{attribute addProperty BoxType "EP9128-0021-0018"}
{attribute addProperty Id "A_0013_EP9128_0021_0019A_0013_EP9128_0021_0019_07EDD1EA4534566.75A_0010_EP9128_0021_0018_2_EP9128_1021EP9128_179A0949162A_0010_EP9128_0021_0018_3_EP9128_2021EP9128_179A0949162"}
{attribute addProperty CRC "2766684775"}
{attribute addProperty SizeInBites "4566"}
{attribute addProperty SizeInBytes "570.75"}
TYPE A_0010_EP9128_0021_0018_A4E84267 EXTENDS EP9128_179A0949 :
STRUCT
	{attribute addProperty Name "A_0013_EP9128_0021_0019"}
	A_0013_EP9128_0021_0019 : A_0013_EP9128_0021_0019_07EDD1EA;
	{attribute addProperty Name "A_0010_EP9128_0021_0018_2_EP9128_1021"}
	A_0010_EP9128_0021_0018_2_EP9128_1021 : EP9128_179A0949;
	{attribute addProperty Name "A_0010_EP9128_0021_0018_3_EP9128_2021"}
	A_0010_EP9128_0021_0018_3_EP9128_2021 : EP9128_179A0949;
END_STRUCT
END_TYPE

(* stored: Version 1.2.0.0, ProductVersion 3.1.4024.9
   DUT A_0010_EP9128_0021_0018_A4E84267: Id {d8fc677a-aa70-4105-83a8-915e457ee4d4} *)
